// SIMATIC S7-200 project (STEP 7-Micro/WIN), CPU 224XP CN REL 02.01

SYMBOL_TABLE 参数
QLJG             VW306    // 强励时间间隔 3-60分钟
DYST             VD326    // 电压爬升时间 0-10S
QLK              VD330    // 强励条件60-90%
QLBS             VD334    // 强励倍数120-180%
QLT              VD338    // 强励时间 10-60s
COSA             VD342    // 整流角限制 10
COSB             VD346    // 逆变角限制 170
DYGD             VD350    // 机端电压给定 0-180%
DLGD             VD354    // 励磁电流给定
GLYS             VD358    // 功率因数给定
                 VD362    // 机端反馈电压
                 VD366    // 励磁反馈电流
SLICI            VD370    // 失磁动作整定  20-100%
GLICI            VD374    // 过励动作整定  80-180%
KGY              VD378    // 空载电压限制 1.0-2.0
KGL              VD382    // 空载电流限制 1.0-2.0
V5               VD386    // 对应5V
V10              VD390    // 对应10V
END_SYMBOL_TABLE

SYMBOL_TABLE 标志
KAIJI            M0.0     // 开机条件标志
                 M0.1     // 开机
CHAOPIN          M0.7     // 超频标志
QSHIBAI          M1.4     // 强励磁失败 离网
END_SYMBOL_TABLE

ORGANIZATION_BLOCK MAIN:OB1
TITLE=介绍
// 这个PLC程序用于控制火力发电厂的发电机励磁系统。通过自动调节励磁电流，确保发电机在空载、并网及负载变化时输出稳定的电压和功率。系统支持恒压、恒流和恒功率因数三种运行模式，通过VW302（0、1、2）选择。
// 项目包括发电机、励磁系统、快熔断器、风机、电压和电流传感器、PLC控制器、触摸屏。
// 系统详解
// 系统支持三种运行模式：恒压、恒流和恒功率因数，操作员可通过运行模式选择灵活切换，切换后开机条件标志置位时进入相应模式。开机时，操作员按下开机按钮，系统在确认无风机故障信号和其他故障信号后启动，开机条件标志置位后进入相应模式。
// 在恒压模式下，系统根据机端电压反馈和机端电压给定，通过PID控制器调整模拟量输出，确保电压稳定；在恒流模式下，依赖励磁电流反馈和励磁电流给定保持电流恒定；在恒功率因数模式下，则根据功率因数反馈进行调节。PID控制中，PID增益始终保持在0.0到1.0之间，避免因参数异常导致系统振荡。
// 为保障安全，程序内置多重保护机制。若检测到快熔断器故障信号，系统立即置位离网信号、电阻接入信号和脉冲封锁信号，同时点亮快熔断器故障指示灯并在延时后触发蜂鸣器提示。若快熔断器故障信号触发，点亮故障指示灯以提示操作员。若机端电压反馈超出空载电压限制，系统检测并在延时后置位过压故障信号；若励磁电流反馈低于失磁动作整定，延时后置位失励磁故障信号，确保故障及时响应。
// 并网运行时并网信号置位，若励磁电流反馈不足，系统进入强励磁模式，调整PID设定值提升电流，但需注意此值应控制在合理范围内以保护设备。若强励磁超时未达要求，置位强励磁失败标志并触发离网信号。并网运行中若检测到故障，离网信号置位以切断电网连接。停机时，按下停机按钮或检测到严重故障，系统执行逆变灭磁，置位脉冲封锁信号和电阻接入信号，确保安全停机。
BEGIN
Network 1
// 正常模式
LD     SM0.0
AW=    VW308, 0
CALL   MAIN0:SBR0
Network 2 // 


// 烘干模式
LD     SM0.0
AW=    VW308, 1
MOVR   V5:VD386, LD0
*R     DLGD:VD354, LD0
MOVR   LD0, VD420
/R     100.0, VD420
CALL   BIAOZHUN2:SBR3
Network 3
// 强励磁
LD     SM0.0
CALL   QIANGLI:SBR2
END_ORGANIZATION_BLOCK

SUBROUTINE_BLOCK MAIN0:SBR0
TITLE=主程序
BEGIN
Network 1
// 参数
LD     SM0.0
CALL   CHANSHU:SBR6
Network 2
// 开机
LD     SM0.0
LD     I0.0
AN     I0.3
AN     I0.4
LD     KAIJI:M0.0
AN     Q1.1
OLD
ALD
=      KAIJI:M0.0
Network 3
// 恒压模式
LD     SM0.0
AW=    VW302, 0
MOVW   AIW0, VW90
MOVR   V5:VD386, LD0
*R     DYGD:VD350, LD0
/R     3200000.0, LD0
MOVR   LD0, VD200
A      KAIJI:M0.0
CALL   PIDGD:SBR8
Network 4
// 恒流模式
LD     SM0.0
AW=    VW302, 1
MOVW   AIW2, VW90
MOVR   V5:VD386, LD4
*R     DLGD:VD354, LD4
/R     3200000.0, LD4
MOVR   LD4, VD200
A      KAIJI:M0.0
CALL   PIDGD:SBR8
Network 5
// 恒功率因数
LD     SM0.0
AW=    VW302, 2
MOVW   AIW4, VW90
A      KAIJI:M0.0
CALL   PIDGD:SBR8
Network 6
// 并网模式 自动转入电流模式
LD     SM0.0
A      I0.6
EU
MOVW   1, VW302
Network 7
// 故障判断
LD     SM0.0
A      KAIJI:M0.0
TON    T32, 20
A      T32
CALL   GUZHANG:SBR5
Network 8
// 故障指示灯           快熔，风机
LD     SM0.0
LPS
A      I0.2
=      Q0.2
LPP
A      I0.3
=      Q0.3
Network 9
// 快熔断停机 封锁脉冲/ 电阻接入/离网
LD     SM0.0
A      I0.2
=      Q1.2
=      Q1.1
=      Q0.0
Network 10
// 停机  快熔断/ 风机短路/过压/失励磁/过励/频率/停机开关
LD     SM0.0
AN     I0.6
A      KAIJI:M0.0
LD     I0.1
O      Q0.6
O      M0.4
O      Q0.5
O      Q0.4
O      M1.0
O      Q0.7
ALD
CALL   MIECI:SBR9
=      M0.1
Network 11
// 并网停机
LD     SM0.0
A      I0.6
A      KAIJI:M0.0
LD     Q0.4
O      Q0.6
ALD
=      Q1.2
=      M1.3
Network 12
// 蜂明器
LD     SM0.0
LD     I0.2
O      I0.3
O      M0.1
O      M1.3
ALD
TON    T102, 300
A      T102
=      Q0.1
Network 30 // 网络标题
// 网络注释
END_SUBROUTINE_BLOCK

SUBROUTINE_BLOCK PIDBIAOZHUN:SBR1
TITLE=逆变角度标准
BEGIN
Network 1 // 网络标题
// 网络注释
LD     SM0.0
MOVW   0, VW318
ROUND  VD416, AC3
DTI    AC3, AC3
MOVW   AC3, VW318
END_SUBROUTINE_BLOCK

SUBROUTINE_BLOCK QIANGLI:SBR2
TITLE=强励控制
BEGIN
Network 1 // 网络标题
// 网络注释
LD     SM0.0
LPS
AN     M1.5
A      I0.6
AW=    VW304, 1
LPS
MOVR   QLK:VD330, LD0
*R     V5:VD386, LD0
MOVW   AIW2, VW316
AENO
CALL   BAIFENBI:SBR4
LPP
AR<    VD394, LD0
LPS
MOVW   1, VW302
MOVW   VW338, LW10
*I     +10, LW10
EU
TOF    T103, LW10
LRD
A      T103
MOVR   QLBS:VD334, VD200
*R     0.05, VD200
LPP
AW=    T103, LW10
AR<    VD394, LD0            //强励磁失败 离网
S      M1.5, 1
=      QSHIBAI:M1.4
LPP
LPS
MOVW   QLJG:VW306, LW12
*I     +600, LW12
A      M1.5
EU
TOF    T104, LW12
LPP
AW=    T104, LW12
R      M1.5, 1
END_SUBROUTINE_BLOCK

SUBROUTINE_BLOCK BIAOZHUN2:SBR3
TITLE=浮点整数化
BEGIN
Network 1 // 网络标题
// 网络注释
LD     SM0.0
ROUND  VD420, AC2
DTI    AC2, AC2
INVW   AC2
INCW   AC2
+I     25600, AC2
MOVW   AC2, AQW0
END_SUBROUTINE_BLOCK

SUBROUTINE_BLOCK BAIFENBI:SBR4
TITLE=百分比参数标准
BEGIN
Network 1 // 网络标题
// 网络注释
LD     SM0.0
MOVW   0, AC1
MOVR   0.0, VD394
ITD    VW316, AC1
DTR    AC1, AC1
*R     100.0, AC1
MOVR   AC1, VD394
END_SUBROUTINE_BLOCK

SUBROUTINE_BLOCK GUZHANG:SBR5
TITLE=限制条件
BEGIN
Network 1 // 网络标题
// 空载过压
LD     SM0.0
AN     I0.6
MOVR   V5:VD386, LD0
*R     KGY:VD378, LD0
MOVW   AIW0, VW316
CALL   BAIFENBI:SBR4
AR>    VD394, LD0
=      M0.2
Network 2
// 过压故障输出延时
LD     SM0.0
AN     I0.6
A      M0.2
TON    T99, 100
A      T99
=      Q0.6
Network 3
// 空载过流/过励
LD     SM0.0
AN     I0.6
LPS
MOVR   V5:VD386, LD4
*R     KGL:VD382, LD4
MOVR   V5:VD386, LD12
*R     GLICI:VD374, LD12
MOVW   AIW2, VW316
CALL   BAIFENBI:SBR4
AR>    VD394, LD4
=      M0.3
LPP
AR>    VD394, LD12
=      M0.6
Network 4
// 空载过流/过励 故障输出延时
LD     SM0.0
AN     I0.6
LPS
A      M0.3
TON    T98, 100
A      T98
=      M0.4
LPP
A      M0.6
TON    T97, 100
A      T97
=      Q0.5
Network 5
// 失磁
LD     SM0.0
MOVR   V5:VD386, LD8
*R     SLICI:VD370, LD8
MOVW   AIW2, VW316
CALL   BAIFENBI:SBR4
AR>    LD8, VD394
=      M0.5
Network 6
// 失磁输出延时
LD     SM0.0
A      M0.5
TON    T36, 100
A      T36
=      Q0.4
Network 7
// 并网限制条件  低电压强励磁限制  过励磁
LD     SM0.0
A      I0.6
AW=    VW304, 1
MOVR   V5:VD386, LD24
*R     QLBS:VD334, LD24
MOVW   AIW2, VW316
CALL   BAIFENBI:SBR4
AR>    VD394, LD24
=      M1.2
Network 8
// 强励磁限制  过励磁输出延时
LD     SM0.0
A      I0.6
A      M1.2
TON    T35, 1
A      T35
=      Q0.6
Network 9
// 频率
LD     SM0.0
LPS
MOVR   V5:VD386, LD16
*R     VD398, LD16
MOVR   V5:VD386, LD20
*R     VD402, LD20
MOVW   AIW4, VW320
CALL   BIAOZHUN:SBR7
AR>    VD410, LD16
=      CHAOPIN:M0.7
LPP
AR>    LD20, VD410
=      M1.1
Network 10
// 高低频延时报警
LD     SM0.0
LPS
A      CHAOPIN:M0.7
TON    T34, 50
A      T34
=      M1.0
LPP
A      M1.1
TON    T33, 50
A      T33
=      Q0.7
END_SUBROUTINE_BLOCK

SUBROUTINE_BLOCK CHANSHU:SBR6
TITLE=参数限制与设定
BEGIN
Network 1 // 网络标题
//  //强励时间间隔
// //电压爬升时间
// //强励条件
//  //强励倍数
// //强励时间
// //机端电压给定
// //励磁电流给定
// //失磁动作整定
//  //过励动作整定
// //空载电压限制
// //空载电流限制
LD     SM0.0
LPS
AW<    QLJG:VW306, 3
MOVW   3, QLJG:VW306
LPP
AW>    QLJG:VW306, 60
MOVW   60, QLJG:VW306
Network 2
LD     SM0.0
LPS
AR<    DYST:VD326, 0.0
MOVR   0.0, DYST:VD326
LRD
AR>    DYST:VD326, 10.0
MOVR   10.0, DYST:VD326
LRD
AR<    QLK:VD330, 60.0
MOVR   60.0, QLK:VD330
LPP
AR>    QLK:VD330, 90.0
MOVR   90.0, QLK:VD330
Network 3
LD     SM0.0
LPS
AR<    QLBS:VD334, 120.0
MOVR   120.0, QLBS:VD334
LRD
AR>    QLBS:VD334, 180.0
MOVR   180.0, QLBS:VD334
LRD
AR<    QLT:VD338, 10.0
MOVR   10.0, QLT:VD338
LPP
AR>    QLT:VD338, 60.0
MOVR   60.0, QLT:VD338
Network 4
LD     SM0.0
LPS
AR<    COSA:VD342, 10.0
MOVR   10.0, COSA:VD342
LRD
AR>    COSA:VD342, 80.0
MOVR   80.0, COSA:VD342
LRD
AR<    COSB:VD346, 80.0
MOVR   80.0, COSB:VD346
LPP
AR>    COSB:VD346, 170.0
MOVR   170.0, COSB:VD346
Network 5
LD     SM0.0
LPS
AR<    DYGD:VD350, 0.0
MOVR   0.0, DYGD:VD350
LRD
AR>    DYGD:VD350, 180.0
MOVR   180.0, DYGD:VD350
LRD
AR<    DLGD:VD354, 0.0
MOVR   0.0, DLGD:VD354
LPP
AR>    DLGD:VD354, 180.0
MOVR   180.0, DLGD:VD354
Network 6
LD     SM0.0
LPS
AR<    SLICI:VD370, 20.0
MOVR   20.0, SLICI:VD370
LRD
AR>    SLICI:VD370, 100.0
MOVR   100.0, SLICI:VD370
LRD
AR<    GLICI:VD374, 80.0
MOVR   80.0, GLICI:VD374
LPP
AR>    GLICI:VD374, 180.0
MOVR   180.0, GLICI:VD374
Network 7
// 空载电流限制
LD     SM0.0
LPS
AR<    KGY:VD378, 100.0
MOVR   100.0, KGY:VD378
LRD
AR>    KGY:VD378, 200.0
MOVR   200.0, KGY:VD378
LRD
AR<    KGL:VD382, 100.0
MOVR   100.0, KGL:VD382
LPP
AR>    KGL:VD382, 200.0
MOVR   200.0, KGL:VD382
Network 8
// 设定/增益
LD     SM0.0
LPS
AR<    VD200, 0.0
MOVR   0.0, VD200
LRD
AR>    VD200, 1.0
MOVR   1.0, VD200
LRD
AR<    VD204, 0.0
MOVR   0.0, VD204
LPP
AR>    VD204, 1.0
MOVR   1.0, VD204
Network 9
// 采样时间/积分
LD     SM0.0
LPS
AR<    VD208, 0.0
MOVR   0.0, VD208
LRD
AR>    VD208, 100.0
MOVR   100.0, VD208
LRD
AR<    VD212, 0.0
MOVR   0.0, VD212
LPP
AR>    VD212, 100.0
MOVR   100.0, VD212
Network 10
// 微分/积分分离
LD     SM0.0
LPS
AR<    VD216, 0.0
MOVR   0.0, VD216
LRD
AR>    VD216, 100.0
MOVR   100.0, VD216
LRD
AR<    VD220, 0.0
MOVR   0.0, VD220
LPP
AR>    VD220, 100.0
MOVR   100.0, VD220
END_SUBROUTINE_BLOCK

SUBROUTINE_BLOCK BIAOZHUN:SBR7
TITLE=整数浮点化
BEGIN
Network 1 // 网络标题
// 网络注释
LD     SM0.0
MOVR   0.0, AC0
MOVR   0.0, VD410
ITD    VW320, AC1
DTR    AC1, AC1
MOVR   AC1, VD410
END_SUBROUTINE_BLOCK

SUBROUTINE_BLOCK PIDGD:SBR8
TITLE=PID给定
BEGIN
Network 1 // 网络标题
// 装载PID参数调用PID中断
// 1、回路设定VD200=VD104
// 2、回路增益VD204=VD112
// 3、回路采样时间VD208=VD116
// 4、积分时间VD212=VD120
// 5、关闭微分作用VD216=VD124
// 6、设定中断定时器时间SMB34=10
// 7、设定中断级别
// 8、开
LD     SM0.0
MOVR   VD200, VD104
MOVR   VD204, VD112
MOVR   VD208, VD116
MOVR   VD212, VD120
MOVR   VD216, VD124
ATCH   PIDKZ:INT0, 10
ENI
END_SUBROUTINE_BLOCK

SUBROUTINE_BLOCK MIECI:SBR9
TITLE=停机完全逆变灭磁
BEGIN
Network 1 // 网络标题
// 网络注释
LD     SM0.0
LPS
EU
TOF    T100, 200
LRD
A      T100
MOVR   COSB:VD346, LD0
*R     145.0, LD0            //逆变
MOVR   LD0, VD420
CALL   BIAOZHUN2:SBR3
LPP
AW=    T100, 200
LPS
EU                           //脉冲封锁
TOF    T101, 10
LRD                          //电阻接入2.5%-20%
A      T101
=      Q1.1
LPP
AW>=   AIW2, 400
AW<=   AIW2, 8000
=      Q0.0
END_SUBROUTINE_BLOCK

INTERRUPT_BLOCK PIDKZ:INT0
TITLE=PID中断控制和输出
BEGIN
Network 1
// //将反馈量实数标准化
// 1、整数变双整数
// 2、双整数变实数
// 3、数值标准化
// 4、标准化的反馈量存入回路表
// 
LD     SM0.0
ITD    VW90, AC0
DTR    AC0, AC0
/R     32000.0, AC0
MOVR   AC0, VD100
PID    VB100, 0
Network 2
// //将PID结果转为模拟量
// 1、输出量送累加器
// 2、数值标准化
// 3、实数变整数
// 4、将数值写AQW0
LD     SM0.0
LPS
MOVR   VD108, AC0
*R     32000.0, AC0
ROUND  AC0, AC0
DTI    AC0, AC0
MOVR   COSA:VD342, LD0
*R     145.0, LD0
MOVR   LD0, VD416
AENO
CALL   PIDBIAOZHUN:SBR1      //输出下限
MOVW   VW318, LW10
LRD
MOVR   COSB:VD346, LD4
*R     145.0, LD4
LRD
MOVR   LD4, VD416
AENO
CALL   PIDBIAOZHUN:SBR1      //输出上限
MOVW   VW318, LW12
LPP
AW>=   AC0, LW10
AW<=   AC0, LW12
INVW   AC0
INCW   AC0
+I     25600, AC0
MOVW   AC0, AQW0
END_INTERRUPT_BLOCK
